(* IEC 61131-3 sources: rust-plc/tests/e2e-deploy/fixtures/test-project, 2 files *)

(* ---- helper.st ---- *)
FUNCTION_BLOCK Accumulator
VAR
    total : INT := 0;
END_VAR
VAR_INPUT
    value : INT;
END_VAR
    total := total + value;
END_FUNCTION_BLOCK

(* ---- main.st ---- *)
PROGRAM Main
VAR
    counter : INT := 0;
    cycle_active : BOOL := TRUE;
END_VAR
    counter := counter + 1;
END_PROGRAM
